TYPE ST_NctProcessData :
STRUCT
	///Process data
	AppData0: USINT;
	AppData1: USINT;
	AppData2: USINT;
	AppData3: USINT;
	AppData4: USINT;
END_STRUCT
END_TYPE

(* stored: Version 1.1.0.1, ProductVersion 3.1.4026.12
   DUT ST_NctProcessData: Id {d109fc8e-628a-0425-3625-11f80082cdbe} *)
